Fanuc KAREL source: ko00095.KL

-- PROVISIONAL review KL for V770-1; original PC SHA256 bdb967abf1a92e035f6114f59b6d28d3fda974adf2ca6cb36d4cf550a08fd076
-- Incomplete behavior may be omitted. Consult companion uncertainty JSON. Do not deploy.
PROGRAM KO00095
%NOLOCKGROUP
BEGIN
  -- UNRESOLVED_PC offsets 5-12; opcodes 9D,23
  -- UNRESOLVED_PC offsets 17-69; opcodes 27,27,49,7E,AD,27,49,7E,AD,22,31,7E,4A
  -- UNRESOLVED_PC offsets 74-78; opcodes 7F
END KO00095
